// TwinCAT 3 PLC project GrabAss
// ProgramVersion: 3.1.4024.12
// libraries:
//   Tc2_MC2, * (Beckhoff Automation GmbH)
//   Tc2_Standard, * (Beckhoff Automation GmbH)
//   Tc2_System, * (Beckhoff Automation GmbH)
//   Tc3_Module, * (Beckhoff Automation GmbH)
// project tree:
//   GVLs/ HAVL.TcGVL
//   / PlcTask.TcTTO
//   POUs/ HorAxisPosCon.TcPOU, MAIN.TcPOU, RunGRAB.TcPOU
// real-time tasks:
//   TASK PlcTask: cycle T#10ms, priority 20, ADS port 350
// motion (NC):
//   TASK NC-Task 1 SAF: cycle T#2ms, priority 4, ADS port 501
//   TASK NC-Task 1 SVB: cycle T#10ms, priority 8, ADS port 511
//   AXIS Axis 1 (id 1)
//     General: UnitName=m
//     Dynamic: AccelerationMaximum=2, DecelerationMaximum=2, Acceleration=0.5, Deceleration=0.5, Jerk=5
//     Velo: RefSearch=0.08, RefSync=0.02, SlowManual=0.1, FastManual=0.3, Maximum=1.00531
//     OtherSettings: AllowMotionCmdToSlave=true, PulseDistancePos=0.005, PulseDistanceNeg=0.005
//     encoder EncType=19
//       EncPara: ScaleFactorNumerator=4.208e-06, MaxCount=#xffffffff
//         SoftEndMinControl: Enable=true, Range=-0.02
//         SoftEndMaxControl: Enable=true, Range=1.5
//         Inc: RefSoftSyncMask=#x00000fff
//     drive DrvType=16
//       DrvPara: MaxCount=#xffffffff, DriveControlDWord=#x00020000
//         Analog: VeloReferenz=1.005309649, TorqueSetpointScale=10, ScaleFactorActTorque=0.1
//         TimeComp: TaskDelayCycles=1
//     controller CtrType=1
//       CtrPara: PriorControlFactor=1
//         Observer: BandWidth=20
// I/O:
//   DEVICE Device 1 (EtherCAT), AmsNetId 5.46.12.154.2.1
//     Term 1 (EK1200) [EK1200-5000 EtherCAT Power supply (2A E-Bus)]
//       Term 2 (EK1110) [EK1110 EtherCAT extension]
//     Drive 3 (N5-2-1) [N5 EtherCAT Drive (CoE)]
// variable links:
//   NC-Task 1 SAF/Axes/Axis 1 <-> Device 1 (EtherCAT)/Drive 3 (N5-2-1)
//     Drive/Inputs/In/nState1 <-> Transmit PDO 1 Mapping Parameter/Statusword
//     Drive/Inputs/In/nState2 <-> Transmit PDO 1 Mapping Parameter/Statusword @bit 8
//     Drive/Inputs/In/nState4 @bit 1 <-> WcState/InputToggle
//     Drive/Inputs/In/nState4 <-> WcState/WcState
//     Drive/Inputs/In/nState5 <-> Transmit PDO 1 Mapping Parameter/Modes of operation display
//     Drive/Outputs/Out/nCtrl1 <-> Receive PDO 1 Mapping Parameter/Controlword
//     Drive/Outputs/Out/nCtrl2 <-> Receive PDO 1 Mapping Parameter/Controlword @bit 8
//     Drive/Outputs/Out/nCtrl5 <-> Receive PDO 1 Mapping Parameter/Modes of operation
//     Drive/Outputs/Out/nDataOut1 <-> Receive PDO 1 Mapping Parameter/Target Position
//     Enc/Inputs/In/nDataIn1 <-> Transmit PDO 1 Mapping Parameter/Position actual value
//     Enc/Inputs/In/nState4 @bit 1 <-> WcState/InputToggle
//     Enc/Inputs/In/nState4 <-> WcState/WcState
//   GrabAss/GrabAss Instance <-> Device 1 (EtherCAT)/Drive 3 (N5-2-1)
//     PlcTask Outputs/MAIN.iMotorDriveSubmodeSelect <-> Receive PDO 1 Mapping Parameter/Motor drive submode select
//   GrabAss/GrabAss Instance <-> NC-Task 1 SAF/Axes/Axis 1
//     PlcTask Inputs/MAIN.axis.NcToPlc <-> Outputs/ToPlc
//     PlcTask Outputs/MAIN.axis.PlcToNc <-> Inputs/FromPlc

CONFIGURATION GrabAss
    RESOURCE PLC ON TwinCAT3
        TASK PlcTask(INTERVAL := T#10ms, PRIORITY := 20);
        PROGRAM MAIN WITH PlcTask : MAIN;
    END_RESOURCE
END_CONFIGURATION

// ---- GVLs/HAVL.TcGVL
{attribute 'qualified_only'}
VAR_GLOBAL
	axis: AXIS_REF;
	axisPower: MC_Power;
	axisMoveAbsolute: MC_MoveAbsolute;
	axisErrorReset: MC_Reset;
	axisReadActualPosition: MC_ReadActualPosition;
	axisMoveManual: MC_Jog;
	
	enable: BOOL := FALSE;
	override: LREAL := 100;
	enableMove: BOOL := FALSE;
	targetPosition: LREAL := 0.1;
	targetVelocity: LREAL := 0.03;
	motorDriveSubmodeSelect AT%Q*:UDINT := 65;
END_VAR

// ---- POUs/MAIN.TcPOU
PROGRAM MAIN
VAR
END_VAR

HorAxisPosCon();

END_PROGRAM

// ---- POUs/HorAxisPosCon.TcPOU
PROGRAM HorAxisPosCon
VAR
	running: BOOL := FALSE;
	busy: BOOL := TRUE;
	done: bool := TRUE;
	
	fbTimer: TON;
	tTimerValue     : TIME := T#5S;
	bStart          : BOOL := TRUE;
	
	reset: BOOL := FALSE;
	
	currentError: UDINT;
	
	start: BOOL := FALSE;
	position: LREAL;
END_VAR

HAVL.axis.ReadStatus();

fbTimer(IN := bStart, PT := tTimerValue);
IF done THEN
	bStart := TRUE;
END_IF

IF start AND NOT(busy) THEN
	HAVL.enable := TRUE;
ELSIF NOT(start) AND NOT(busy) THEN
	HAVL.enable := FALSE;
END_IF

HAVL.axisPower(
	Axis:= HAVL.axis,
	Enable:= HAVL.enable,
	Enable_Positive:= HAVL.enable,
	Enable_Negative:= HAVL.enable,
	Override:= HAVL.override,
	BufferMode:= ,
	Options:= ,
	Status=> running,
	Busy=> ,
	Active=> ,
	Error=> ,
	ErrorID=> currentError
);

HAVL.axisMoveAbsolute(
	Axis:= HAVL.axis,
	Execute:= HAVL.enableMove,
	Position:= HAVL.targetPosition,
	Velocity:= HAVL.targetVelocity,
	Acceleration:= ,
	Deceleration:= ,
	Jerk:= ,
	BufferMode:= ,
	Options:= ,
	Done=> done,
	Busy=> busy,
	Active=> ,
	CommandAborted=> ,
	Error=> ,
	ErrorID=> currentError 
);

IF NOT(busy) AND NOT(HAVL.enableMove)AND running AND HAVL.enable AND fbTimer.Q THEN
	HAVL.enableMove := TRUE;
	bStart := FALSE;
	IF HAVL.targetPosition = 0 THEN
		HAVL.targetPosition := 0.1;
	ELSE
		HAVL.targetPosition := 0;
	END_IF
END_IF

IF busy AND HAVL.enableMove THEN
	HAVL.enableMove := FALSE;
END_IF

HAVL.axisErrorReset(Axis := HAVL.axis, Execute := reset, Done =>, Error =>, ErrorID => currentError);

HAVl.axisReadActualPosition(Axis := HAVL.axis, Enable := busy, Valid=>, Busy=>, Error=>, ErrorID=>, Position=> position);

END_PROGRAM

// ---- POUs/RunGRAB.TcPOU
PROGRAM RunGRAB
VAR
END_VAR

END_PROGRAM
